# EPICS substitutions: agilent53210App/Db/agilent53210aEX.substitutions
# Agilent 53210A frequency counter
file agilent53210a.template
{
pattern {  DEVICE        , PORT    , SCAN  }
        {  OSC:LR20:20: , "agilFC" , "1 second"      }
}

# DEVICE: device name
# PORT: asyn communication port
# SCAN: refrash rate
